// TIA Portal V21 export
TYPE "motorAlm"
   STRUCT
      fault : Bool;   // motor protection tripped or no signal
      falseFbFwd : Bool;
      falseFbRev : Bool;
      stickingFwd : Bool;
      stickingRev : Bool;
      badCmd : Bool;   // Both fwd and rev input present at the same time
      noFbFwd : Bool;
      noFbRev : Bool;
      badOut : Bool;
      extStop : Bool := false;
      stepErr : Bool := false;
      bit11 : Bool := false;
      bit12 : Bool := false;
      bit13 : Bool := false;
      bit14 : Bool := false;
      bit15 : Bool := false;
   END_STRUCT;
END_TYPE
